{attribute 'GeneratedUsingTerminal: EK1100-0000-0018'}
{attribute addProperty BoxType "EK1100-0000-0018"}
{attribute addProperty Id "Beckhoff_EP1xxxEK1122Beckhoff_EP1xxxEK1122_3357DBA91740"}
{attribute addProperty CRC "1634739946"}
{attribute addProperty Size "1740"}
TYPE Beckhoff_EP1xxx_617026EA EXTENDS EK1100_1FC0878B :
STRUCT
	{attribute addProperty Name "Beckhoff_EP1xxxEK1122"}
	Beckhoff_EP1xxxEK1122 : Beckhoff_EP1xxxEK1122_3357DBA9;
END_STRUCT
END_TYPE

(* stored: Version 1.2.0.0, ProductVersion 3.1.4024.9
   DUT Beckhoff_EP1xxx_617026EA: Id {8022e5ef-42ce-4464-87cd-d7269dca7f88} *)
